// TIA Portal V20 export
TYPE "typeTopTapeIdleTimeHmiInterface"
// stored: Access Published, Namespace Unit1.Em3
   STRUCT
      currentCount : Time;
      processCount : Time := T#0ms;
   END_STRUCT;
END_TYPE
